TYPE EcCoeSdo_Ctrl_typ :
	STRUCT
		Input	: EcCoeSdo_Input_typ ;
		Output	: EcCoeSdo_Output_typ ;
	END_STRUCT
END_TYPE

(* stored: Version 1.1.0.1, ProductVersion 3.1.4024.3
   DUT EcCoeSdo_Ctrl_typ: Id {e9db7892-d480-037f-07b3-b9054caf14f4} *)
